(* =========================================================================================================================
   Base FB/class
   =========================================================================================================================
   Description:
   This base class contains/provides some basic functionalities:
   - implementation of the interface "I_Sample"
   - basic implementation of the method called "Calculate" (in this case, the sum of two input parameters is returned)
   - ID handling via a property and a local variable to provide an object of this class with an ID
        - nObjectID.Get to read the ID of an object
        - nObjectID.Set to write the ID of an object
   ========================================================================================================================= *)
FUNCTION_BLOCK FB_Sample_Base IMPLEMENTS I_Sample
VAR
	nID		: INT;
END_VAR

METHOD Calculate : INT
VAR_INPUT
	nIn1	: INT;
	nIn2	: INT;
END_VAR
Calculate := nIn1 + nIn2;
END_METHOD

PROPERTY nObjectID : INT
GET
nObjectID := nID;
END_GET
SET
IF nObjectID > 0 THEN
	 nID := nObjectID;
END_IF
END_SET
END_PROPERTY

END_FUNCTION_BLOCK

(* stored: Version 1.1.0.1, ProductVersion 3.1.4024.0
   POU FB_Sample_Base: Id {3bd7b26d-f8ab-450c-ae2f-8ae59a2d67a3}, SpecialFunc None
   Method Calculate: Id {00d54ebb-025d-42b4-af18-944c5fc0a7ce}
   Property nObjectID: Id {84944678-0099-4b7f-b981-1d96e05b5e55}
   Get Get: Id {63ed9b03-7f0b-44c4-91c4-df706795149c}
   Set Set: Id {c9a0260a-7617-4465-969d-208aa1cec17f} *)
